FUNCTION TryConvert_TOD_TO_TIME : BOOL
VAR_INPUT
	in : TOD;
	out : REFERENCE TO TIME;
END_VAR

out := TOD_TO_TIME(in);
TryConvert_TOD_TO_TIME := TRUE;

END_FUNCTION

(* stored: Version 1.1.0.1, ProductVersion 3.1.4024.12
   POU TryConvert_TOD_TO_TIME: Id {f3678dce-1413-44b7-b408-5ad41fdc761a}, SpecialFunc None *)
